PROGRAM MAIN
VAR
	step : UINT;
	fbChainController : FB_ChainController;
	fbChain1 : FB_TestChain1;
	fbChain2 : FB_TestChain2;
END_VAR

fbChain1(io_fbChainController := fbChainController);
fbChain2(io_fbChainController := fbChainController);

fbChain1.define(uiChainNumber := 1, sChainName := 'fbChain1');
fbChain2.define(uiChainNumber := 2, sChainname := 'fbChain2');

CASE step OF

	10: 
		fbChainController
			.addChain(fbChain1)
			.addChain(fbChain2);
		
		fbChain1.cmdIgnite();
		fbChain2.cmdIgnite();	
		step := 20;
		
	20:
	
		
END_CASE

END_PROGRAM

(* stored: Version 1.1.0.1, ProductVersion 3.1.4024.0
   POU MAIN: Id {358f7823-9894-4896-a8c5-c2f64c09a379}, SpecialFunc None *)
